# EPICS StreamDevice protocol: protocols/acq480.proto
Terminator = LF;
ExtraInput = Ignore;

setInvert {
	out "acq480_setInvert \$1 %d";
	in;
}

setGain {
	out "acq480_setGain \$1 %d";
	in;
}

setHPF {
# channel enable K   enable = K!=0
	out "acq480_setHiPassFilter \$1 %d %d";
	in;
}

setLFNS {
	out "acq480_setLFNS \$1 %d";
	in;
}

setFIR {
	# odd-chan for Custom : TODO. Custom: TODO
	out "acq480_setDecimationFilter \$1 %d 0";
	in;
}

# T50R_[1-8] or T50R (global) value 0 or 1
setT50R {
	out "T50R\$1 %d";
	in;
}

getT50R {
	out "T50R\$1";
	in "%d";
}

# getTrain : unsolicited data on 4320+SITE
getTrain {
	in "%d";
}

getJC {
	out "JC_\$1";
	in "%d";
}

getLOTI {
	out "acq480_loti";
	in "%d";
}

get2LM {
	out "acq480_two_lane_mode";
	in "%d";
}

getStack {
    out "acq480_stack";
    in "%s";
}

setStack {
       out "acq480_stack %s";
         in;
}
